// TwinCAT 3 PLC project WalslijnPLC
// ProgramVersion: 3.1.4023.0
// libraries:
//   Tc2_Standard, * (Beckhoff Automation GmbH)
//   Tc2_System, * (Beckhoff Automation GmbH)
//   Tc3_Module, * (Beckhoff Automation GmbH)
// project tree:
//   DUTs/Parameters/Continu Walsen/ ENUM_CR_RollingConfiguration.TcDUT, ENUM_CR_TemperatureMode.TcDUT, ST_CR_Coil.TcDUT, ST_CR_CW.TcDUT, ST_CR_Parameters.TcDUT
//   DUTs/Parameters/Discontinu  hot rolling/ ENUM_DCR_RollStand.TcDUT, ST_DHR_Parameters.TcDUT, ST_DHR_ParameterStand.TcDUT, ST_DHR_ProgramOptions.TcDUT, ST_DHR_Rollingschedule_Entry.TcDUT
//   DUTs/Parameters/Discontinu cold rolling/ ST_DCR_Parameters.TcDUT, ST_DCR_ProgramOptions.TcDUT
//   DUTs/Parameters/FDC/ ST_FDC_Parameters.TcDUT
//   DUTs/Parameters/Generic/ ENUM_CoolingMethod.TcDUT, ENUM_FirstPass.TcDUT, ST_RollingConditions.TcDUT, ST_SampleParameters.TcDUT
//   DUTs/Parameters/Logging/ ST_AcquisitionSelection.TcDUT, ST_LogStandard.TcDUT
//   / PlcTask.TcTTO
//   POUs/ MAIN.TcPOU
//   VISUs/ GVL_Visu.TcGVL

CONFIGURATION WalslijnPLC
    RESOURCE PLC ON TwinCAT3
        TASK PlcTask(INTERVAL := T#10ms, PRIORITY := 20);
        PROGRAM MAIN WITH PlcTask : MAIN;
    END_RESOURCE
END_CONFIGURATION

// ---- DUTs/Parameters/Continu Walsen/ENUM_CR_RollingConfiguration.TcDUT
{attribute 'qualified_only'}
{attribute 'strict'}
TYPE ENUM_CR_RollingConfiguration :
(
	CW2 := 0,//CW2 default
	CW1 := 1,
	DualStand := 3
);
END_TYPE

// ---- DUTs/Parameters/Continu Walsen/ENUM_CR_TemperatureMode.TcDUT
{attribute 'qualified_only'}
{attribute 'strict'}
TYPE ENUM_CR_TemperatureMode :
(
	hot := 0,
	cold :=1
);
END_TYPE

// ---- DUTs/Parameters/Continu Walsen/ST_CR_Coil.TcDUT
TYPE ST_CR_Coil :
STRUCT
	diameter			: REAL;		//start diameter voor proef in mm		
	stripThickness 		: REAL;		//mm
	stripWidth			: REAL;		//mm
	
END_STRUCT
END_TYPE

// ---- DUTs/Parameters/Continu Walsen/ST_CR_CW.TcDUT
TYPE ST_CR_CW :
STRUCT
	rollGap		: REAL;		// mm
	rollSpeed	: REAL;		// m/s
	acc			: REAL;		// m/s³
	tensionAfw	: REAL;		//trekspanning in N/mm² TODO bij dual stand?
	tensionOpw	: REAL;		//trekspanning in N/mm²	TODO	bij dual stand?

END_STRUCT
END_TYPE

// ---- DUTs/Parameters/Continu Walsen/ST_CR_Parameters.TcDUT
TYPE ST_CR_Parameters :
STRUCT
	rollingConfiguration	: ENUM_CR_RollingConfiguration;
	coil					: ST_CR_Coil;
	temperatureMode			: ENUM_CR_TemperatureMode;
END_STRUCT
END_TYPE

// ---- DUTs/Parameters/Discontinu  hot rolling/ENUM_DCR_RollStand.TcDUT
{attribute 'qualified_only'}
{attribute 'strict'}
TYPE ENUM_DCR_RollStand :
(
	CW2 	:= 0,	//enkel wals 2, default
	CW1 	:= 1	//enkel wals 1
);
END_TYPE

// ---- DUTs/Parameters/Discontinu  hot rolling/ST_DHR_Parameters.TcDUT
TYPE ST_DHR_Parameters :
STRUCT
	sampleParameters		: ST_SampleParameters;
	rollingConditions		: ST_RollingConditions;
	rollingSchedule			: ARRAY[0..14] OF ST_DHR_Rollingschedule_Entry;
	parametersStandCw1		: ST_DHR_ParameterStand;
	parametersStandCw2		: ST_DHR_ParameterStand;
	{info 'TODO: implmement logging config data'} 
	acquisitionSelection	: ST_AcquisitionSelection;
	programOptions			: ST_DHR_ProgramOptions;
	
END_STRUCT
END_TYPE

// ---- DUTs/Parameters/Discontinu  hot rolling/ST_DHR_ParameterStand.TcDUT
TYPE ST_DHR_ParameterStand :
STRUCT
	firstPass				: ENUM_FirstPass;
	changeRotationEachPass 	: BOOL:=TRUE;
	minForceForNextPass		: REAL:=20.0;		// ton
	rollingSpeed			: REAL:=33.0;//rpm (voor discontinu)
END_STRUCT
END_TYPE

// ---- DUTs/Parameters/Discontinu  hot rolling/ST_DHR_ProgramOptions.TcDUT
TYPE ST_DHR_ProgramOptions :
STRUCT
	automaticEndAcquisition			: BOOL;		//logging automatisch stoppen bij einde proef,indien niet geselecteerd moet operator de logging beeindigen
	rollThickBlocksOnCw2			: BOOL;		//ipv eerst draaizin te wijzigen, walsspleet zakken en dan pas draaizin wijzigen
END_STRUCT
END_TYPE

// ---- DUTs/Parameters/Discontinu  hot rolling/ST_DHR_Rollingschedule_Entry.TcDUT
TYPE ST_DHR_Rollingschedule_Entry :
STRUCT
	rollGap 		: REAL;	//mm
	reduction		: REAL;	//%
	Temperature 	: REAL; //°C
	stand			: ENUM_DCR_RollStand;	//keuze wals(en)
	
END_STRUCT
END_TYPE

// ---- DUTs/Parameters/Discontinu cold rolling/ST_DCR_Parameters.TcDUT
TYPE ST_DCR_Parameters :
STRUCT
	sampleParameters	: ST_SampleParameters;
	programOptions		: ST_DCR_ProgramOptions;
END_STRUCT
END_TYPE

// ---- DUTs/Parameters/Discontinu cold rolling/ST_DCR_ProgramOptions.TcDUT
TYPE ST_DCR_ProgramOptions :
STRUCT
	rollingSpeed			: REAL;		//snelheid van wals in tr/min
	forceToReleaseSample	: REAL;		//gewicht in ton voor detectie van het stuk
	timeTableCanMoveBack	: REAL;		//tijd in seconden dat de tafel terug rijdt, bij afwezigheid van eindeloop
	tableHorizontalPos		: REAL;		//analoge positiemeting of terugkoppeling cilinder (momenteel afwezig)
	adaptRollGapAuto		: BOOL;		//automatisch roll gap verkleinen
	adaptationToRollGap		: REAL;		//indien adapt rollgap is geselecteerd, roll gap verkleinen met deze waarde in mm
	nrOfEqualSamples		: USINT;	//hoeveel keer hetzelfde product door de walsspleet duwen
END_STRUCT
END_TYPE

// ---- DUTs/Parameters/FDC/ST_FDC_Parameters.TcDUT
TYPE ST_FDC_Parameters :
STRUCT
	klepModule1			: REAL;		//procentueel 0..100
	klepModule2			: REAL;		//procentueel 0..100
	klepModule3			: REAL;		//procentueel 0..100
	klepModule4			: REAL;		//procentueel 0..100
	frequentiePomp		: REAL;		//RPM
	bankKeuze 			: ENUM_BANKKEUZE;
	snelheidPinchRolss	: REAL;		// m/s
	tijdVooruitAchteruit: REAL;		//	seconden
END_STRUCT
END_TYPE

// ---- DUTs/Parameters/Generic/ENUM_CoolingMethod.TcDUT
{attribute 'qualified_only'}
{attribute 'strict'}
TYPE ENUM_CoolingMethod :
(
	fdc := 0,
	laminair := 1
);
END_TYPE

// ---- DUTs/Parameters/Generic/ENUM_FirstPass.TcDUT
{attribute 'qualified_only'}
{attribute 'strict'}
TYPE ENUM_FirstPass :
(
	Left := 1,
	Right:=0//default
);
END_TYPE

// ---- DUTs/Parameters/Generic/ST_RollingConditions.TcDUT
TYPE ST_RollingConditions :
STRUCT
	temperature		: REAL;
	coolingMethod	: ENUM_CoolingMethod;
	fdcParameters	: ST_FDC_Parameters;
END_STRUCT
END_TYPE

// ---- DUTs/Parameters/Generic/ST_SampleParameters.TcDUT
TYPE ST_SampleParameters :
STRUCT
	thickness			: REAL;
	width				: REAL;
	length				: REAL;
END_STRUCT
END_TYPE

// ---- DUTs/Parameters/Logging/ST_AcquisitionSelection.TcDUT
TYPE ST_AcquisitionSelection :
STRUCT
	
END_STRUCT
END_TYPE

// ---- DUTs/Parameters/Logging/ST_LogStandard.TcDUT
TYPE ST_LogStandard :
STRUCT
	bEnable		: BOOL;		//logging in of uitschakelen
	nSampleRate	: INT;		//snelheid datalog in hz
	bBufferVol	: BOOL;		//buffer is vol
	
END_STRUCT
END_TYPE

// ---- VISUs/GVL_Visu.TcGVL
{attribute 'qualified_only'}
VAR_GLOBAL
	
	DHR_RollingSchedule 	: ST_DHR_Rollingschedule_Entry;

END_VAR

// ---- POUs/MAIN.TcPOU
PROGRAM MAIN
VAR
END_VAR

END_PROGRAM
